FUNCTION_BLOCK CU050ExampleCompositComponent EXTENDS TcoCore.TcoComponent
VAR_INPUT
END_VAR
VAR_OUTPUT
END_VAR
VAR
END_VAR

END_FUNCTION_BLOCK

(* stored: Version 1.1.0.1
   POU CU050ExampleCompositComponent: Id {02a723f5-4be0-47f3-9ef7-13d5d0b6f3fe}, SpecialFunc None *)
